// TIA Portal V20 export
DATA_BLOCK "BK02"   // DB299
// stored: MemoryReserve 100
   VAR
      "X10-1 JR OUT P&P1 Z-AXIS LIMIT SENSOR(-)" : Bool;
      "X10-2 JR OUT P&P1 Z-AXIS HOME SENSOR" : Bool;
      "X12-1 JR OUT P&P1 Z-AXIS LIMIT SENSOR(+)" : Bool;
      "X12-2 JR OUT P&P1 STACK DETECT SENSOR" : Bool;
      "X14-1 JR OUT P&P1 CLAMP OPEN" : Bool;
      "X14-2 JR OUT P&P1 CLAMP CLOSE" : Bool;
      "X16-1 JR OUT P&P1 CLAMP OPEN/CLOSE PRESSURE SENSOR" : Bool;
      "X16-2 JR OUT P&P1 Z-AXIS SAFETY PIN LOADING SENSOR" : Bool;
   END_VAR
BEGIN
END_DATA_BLOCK
